Staubli VAL3: Test_project1.pjx

Parameters version=s7.7.1 stackSize=5000 millimeterUnit=true
Program file=start.pgx
Program file=stop.pgx
Data file=Test_project1.dtx
